// TIA Portal V20 export
VAR_GLOBAL   // PLC tag table "Output Machine"
END_VAR
